Yaskawa INFORM job: MASTER_SCIANA_WYPYCH_V19B_V20.JBI

/JOB
//NAME MASTER_SCIANA_WYPYCH_V19B_V20
///FOLDERNAME KRIS-SCIANA
//POS
///NPOS 34,34,34,0,0,0
///TOOL 0
///POSTYPE PULSE
///PULSE
C00000=-1892,-154570,-122283,86345,27128,74017
C00001=16372,13851,-28345,29847,65698,81079
C00002=16372,13851,-28345,29847,65698,81079
C00003=-134924,-99688,-53786,-66204,70242,24091
C00004=-133006,-99325,-53672,-65896,71493,24318
C00005=-176695,-87708,-37155,-93511,17137,90947
///LIMIT ON
C00006=2742,93585,3795,185755,-92976,161895
C00007=-47810,-164401,-99395,208800,-37060,140059
C00008=-25008,-164401,-99395,208800,-37060,140059
C00009=-139066,-167433,-73920,224964,-65133,122755
C00010=-202120,-71729,-52474,305639,61776,72027
C00011=-222921,-68261,-41537,328835,35764,57721
C00012=-205545,-13917,-16977,340291,79502,59779
C00013=-51501,-125812,-64176,358566,23911,21493
C00014=-32622,-30733,-32179,366302,52491,46231
C00015=-9205,87202,7510,375899,87940,76916
C00016=2742,93585,3795,369870,92976,80039
C00017=-47810,-164401,-99395,392915,37060,58203
C00018=-144334,-114745,-52703,304673,32943,59562
C00019=-212224,-89590,-44081,273617,-21895,86132
C00020=-207912,-39796,-25198,187574,-43757,76150
///LIMIT OFF
C00021=-58328,-62854,-83035,171858,-105078,80127
C00022=-2116,91349,41546,171927,-94395,4477
C00023=-57689,-145217,-94647,174172,-82657,-76372
C00024=-142514,-145217,-94647,174172,-82657,-76372
C00025=-241426,-87690,-46527,89385,7785,2283
C00026=-57689,-145217,-94647,174172,-82657,-76372
C00027=-57689,-145217,-94647,174172,-82657,-76372
C00028=-57689,-145217,-94647,174172,-82657,-76372
C00029=-57689,-145217,-94647,174172,-82657,-76372
///LIMIT ON
C00030=-112096,42070,53628,161176,-60133,-114833
C00031=-80414,54958,78135,193534,-37345,-120618
///LIMIT OFF
C00032=-57689,-145217,-94647,174172,-82657,-76372
///LIMIT ON
C00033=110791,-145217,-94647,190147,-98637,-76372
///LIMIT OFF
BC00000=390791,296,950124
BC00001=238537,627,1021817
BC00002=238537,627,1021817
BC00003=367330,15,898279
BC00004=313789,192941,898279
BC00005=372904,15,924730
BC00006=125260,579,1075155
BC00007=359561,7033,947246
BC00008=314070,7033,947246
BC00009=332820,8933,909582
BC00010=369083,12607,836740
BC00011=370294,12730,834306
BC00012=398174,15,901788
BC00013=294629,148,987790
BC00014=289123,406,1026786
BC00015=125260,726,1075157
BC00016=125260,579,1075155
BC00017=359561,7033,947246
BC00018=359585,15,920251
BC00019=357379,559,901559
BC00020=345218,15,962257
BC00021=264602,1732,1075157
BC00022=125260,1732,1075157
BC00023=359227,7883,960834
BC00024=359227,7883,828289
BC00025=361648,8930,829503
BC00026=359227,7883,960834
BC00027=359227,7883,960834
BC00028=359227,7883,960834
BC00029=359227,7883,960834
BC00030=256146,29489,833209
BC00031=208048,48289,905788
BC00032=359227,7883,960834
BC00033=359227,7883,877534
EC00000=1,-1
EC00001=1,-1
EC00002=1,-1
EC00003=1,-1
EC00004=-798161,-556479
EC00005=1,-1
EC00006=1,-1
EC00007=1,-1
EC00008=1,-1
EC00009=1,-1
EC00010=1,-1
EC00011=1,-1
EC00012=1,-1
EC00013=1,-1
EC00014=1,-1
EC00015=1,-1
EC00016=1,-1
EC00017=1,-1
EC00018=1,-1
EC00019=1,-1
EC00020=0,0
EC00021=1,-1
EC00022=1,-1
EC00023=2,-1
EC00024=2,-1
EC00025=2,-1
EC00026=2,-1
EC00027=2,-1
EC00028=2,-1
EC00029=2,-1
EC00030=-798156,-556475
EC00031=-798156,-556475
EC00032=2,-1
EC00033=2,-1
//INST
///DATE 2023/12/20 15:47
///ATTR SC,RW
///GROUP1 RB1,BS1
///GROUP2 ST1
NOP
DOUT OG#(198) 0
WAIT IG#(198)=0
MOVJ C00000 BC00000 VJ=20.00  +MOVJ EC00000 VJ=20.00
MOVJ C00001 BC00001 VJ=50.00  +MOVJ EC00001 VJ=50.00
CALL JOB:CLEAN-R1_LONG
MOVJ C00002 BC00002 VJ=30.00  +MOVJ EC00002 VJ=30.00
MOVJ C00003 BC00003 VJ=50.00  +MOVJ EC00003 VJ=50.00
MOVJ C00004 BC00004 VJ=50.00  +MOVJ EC00004 VJ=50.00
WAIT SOUT#(57)=ON
DOUT OG#(198) 1
WAIT IG#(198)=1
'------------------
CALL JOB:R1_W09,10(-90,-90)
'------------------
DOUT OG#(198) 2
WAIT IG#(198)=2
MOVJ C00005 BC00005 VJ=50.00  +MOVJ EC00005 VJ=50.00
CALL JOB:CLEAN-R1_LONG
MOVJ C00006 BC00006 VJ=50.00  +MOVJ EC00006 VJ=50.00
MOVJ C00007 BC00007 VJ=50.00  +MOVJ EC00007 VJ=50.00
MOVJ C00008 BC00008 VJ=50.00  +MOVJ EC00008 VJ=50.00
MOVJ C00009 BC00009 VJ=50.00  +MOVJ EC00009 VJ=50.00
MOVJ C00010 BC00010 VJ=50.00  +MOVJ EC00010 VJ=50.00
MOVJ C00011 BC00011 VJ=50.00  +MOVJ EC00011 VJ=50.00
DOUT OG#(198) 3
WAIT IG#(198)=3
'------------------
CALL JOB:R1_W5(0,0)
'------------------
DOUT OG#(198) 4
WAIT IG#(198)=4
MOVJ C00012 BC00012 VJ=50.00  +MOVJ EC00012 VJ=50.00
MOVJ C00013 BC00013 VJ=50.00  +MOVJ EC00013 VJ=50.00
MOVJ C00014 BC00014 VJ=50.00  +MOVJ EC00014 VJ=50.00
MOVJ C00015 BC00015 VJ=50.00  +MOVJ EC00015 VJ=50.00
CALL JOB:CLEAN-R1_LONG
MOVJ C00016 BC00016 VJ=50.00  +MOVJ EC00016 VJ=50.00
MOVJ C00017 BC00017 VJ=50.00  +MOVJ EC00017 VJ=50.00
MOVJ C00018 BC00018 VJ=50.00  +MOVJ EC00018 VJ=50.00
DOUT OG#(198) 5
WAIT IG#(198)=5
'------------
CALL JOB:R1_W7(0,0)
'------------
DOUT OG#(198) 6
WAIT IG#(198)=6
MOVJ C00019 BC00019 VJ=50.00  +MOVJ EC00019 VJ=50.00
'------------
CALL JOB:R1_W09(-90,-90)
'------------
PAUSE
MOVJ C00020 BC00020 VJ=30.00  +MOVJ EC00020 VJ=30.00
MOVJ C00021 BC00021 VJ=30.00  +MOVJ EC00021 VJ=0.78
MOVJ C00022 BC00022 VJ=30.00  +MOVJ EC00022 VJ=0.78
CALL JOB:CLEAN-R1_LONG
MOVJ C00023 BC00023 VJ=30.00  +MOVJ EC00023 VJ=0.78
MOVJ C00024 BC00024 VJ=30.00  +MOVJ EC00024 VJ=0.78
MOVJ C00025 BC00025 VJ=30.00  +MOVJ EC00025 VJ=0.78
CALL JOB:R1_W5(0,0)
MOVJ C00026 BC00026 VJ=30.00  +MOVJ EC00026 VJ=0.78
CALL JOB:CLEAN-R1_LONG
MOVJ C00027 BC00027 VJ=30.00  +MOVJ EC00027 VJ=0.78
CALL JOB:R1_W7(0,0)
MOVJ C00028 BC00028 VJ=30.00  +MOVJ EC00028 VJ=0.78
CALL JOB:CLEAN-R1_LONG
MOVJ C00029 BC00029 VJ=30.00  +MOVJ EC00029 VJ=0.78
CALL JOB:R1_W9
MOVJ C00030 BC00030 VJ=30.00  +MOVJ EC00030 VJ=0.78
CALL JOB:R1_W10
MOVJ C00031 BC00031 VJ=30.00  +MOVJ EC00031 VJ=0.78
MOVJ C00032 BC00032 VJ=30.00  +MOVJ EC00032 VJ=0.78
MOVJ C00033 BC00033 VJ=30.00  +MOVJ EC00033 VJ=0.78
CALL JOB:R1_W14
END
